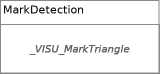
VISUALIZATION _VISU_MarkDefinition_View  // 160x74
VAR_IN_OUT
	mInst : FB_MarkDefinition;
  xScale : UDINT;
END_VAR
    Frame (0,24 160x50), invisible if: NOT mInst.sMarkDef[1].sState.bShow
        shows _VISU_MarkTriangle(mInst := mInst.sMarkDef[1])
        p3560616238: mInst.sMarkDef[1].sState.nMove*xScale
    Frame (0,24 160x50), invisible if: NOT mInst.sMarkDef[2].sState.bShow
        shows _VISU_MarkTriangle(mInst := mInst.sMarkDef[2])
        p3560616238: mInst.sMarkDef[2].sState.nMove*xScale
    Frame (0,24 160x50), invisible if: NOT mInst.sMarkDef[3].sState.bShow
        shows _VISU_MarkTriangle(mInst := mInst.sMarkDef[3])
        p3560616238: mInst.sMarkDef[3].sState.nMove*xScale
    Frame (0,24 160x50), invisible if: NOT mInst.sMarkDef[6].sState.bShow
        shows _VISU_MarkTriangle(mInst := mInst.sMarkDef[6])
        p3560616238: mInst.sMarkDef[6].sState.nMove*xScale
    Frame (0,24 160x50), invisible if: NOT mInst.sMarkDef[4].sState.bShow
        shows _VISU_MarkTriangle(mInst := mInst.sMarkDef[4])
        p3560616238: mInst.sMarkDef[4].sState.nMove*xScale
    Frame (0,24 160x50), invisible if: NOT mInst.sMarkDef[5].sState.bShow
        shows _VISU_MarkTriangle(mInst := mInst.sMarkDef[5])
        p3560616238: mInst.sMarkDef[5].sState.nMove*xScale
    Frame (0,24 160x50), invisible if: NOT mInst.sMarkDef[7].sState.bShow
        shows _VISU_MarkTriangle(mInst := mInst.sMarkDef[7])
        p3560616238: mInst.sMarkDef[7].sState.nMove*xScale
    Frame (0,24 160x50), invisible if: NOT mInst.sMarkDef[10].sState.bShow
        shows _VISU_MarkTriangle(mInst := mInst.sMarkDef[10])
        p3560616238: mInst.sMarkDef[10].sState.nMove*xScale
    Frame (0,24 160x50), invisible if: NOT mInst.sMarkDef[8].sState.bShow
        shows _VISU_MarkTriangle(mInst := mInst.sMarkDef[8])
        p3560616238: mInst.sMarkDef[8].sState.nMove*xScale
    Frame (0,24 160x50), invisible if: NOT mInst.sMarkDef[9].sState.bShow
        shows _VISU_MarkTriangle(mInst := mInst.sMarkDef[9])
        p3560616238: mInst.sMarkDef[9].sState.nMove*xScale
    Rectangle (0,0 120x20), "MarkDetection"
END_VISUALIZATION

(* stored: Version 1.1.0.1, ProductVersion 3.1.4024.11
   Visu _VISU_MarkDefinition_View: Id {964d4f37-41f3-4ee5-9c3a-9185ae40a3ac} *)
